Staubli VAL3: stop.pgx

program stop()
begin
  if workingMode()==3
    disablePower()
  endIf
  // -- kill other running task or else nothing will end (?)
  taskKill("doAirexTask")
  taskKill("doModulesTask")
end
